// TwinCAT 3 PLC project Test
// ProgramVersion: 3.1.4022.4
// libraries:
//   Tc2_Standard, * (Beckhoff Automation GmbH)
//   Tc2_System, * (Beckhoff Automation GmbH)
//   Tc3_Module, * (Beckhoff Automation GmbH)
//   Marquee,0.5,HiJack Automation
// project tree:
//   FBs/ FB_SignalHandling.TcPOU
//   GVLs/ GVL_General.TcGVL, GVL_Machine.TcGVL, GVL_SignalHanlding.TcGVL, HardwareInput.TcDUT, HardWareIO.TcDUT, HardwareOutput.TcDUT, MachineMode.TcDUT
//   / PlcTask.TcTTO
//   POUs/ LampControl.TcPOU, LinkHWIO.TcPOU, LinkUI.TcPOU, MAIN.TcPOU, ModeManger.TcPOU, SignalHandler.TcPOU
// real-time tasks:
//   TASK PlcTask: cycle T#10ms, priority 20, ADS port 350
// I/O:
//   DEVICE Device 2 (EtherCAT), AmsNetId 192.168.1.105.3.1
//     Term 1 (EK1814) [EK1814 EtherCAT IO-Coupler  (1A E-Bus, 4 Ch. Dig. In, 3ms, 4 Ch. Dig. Out 24V, 0,5A)]
// variable links:
//   Test/Test Instance <-> Device 2 (EtherCAT)/Term 1 (EK1814)
//     PlcTask Inputs/GVL_Machine.HWIO.HWInput.PauseBtn <-> Channel 3/Input
//     PlcTask Inputs/GVL_Machine.HWIO.HWInput.StartBtn <-> Channel 1/Input
//     PlcTask Inputs/GVL_Machine.HWIO.HWInput.StopBtn <-> Channel 2/Input
//     PlcTask Outputs/GVL_Machine.HWIO.HWOutput.Lamp01 <-> Channel 5/Output
//     PlcTask Outputs/GVL_Machine.HWIO.HWOutput.Lamp02 <-> Channel 6/Output
//     PlcTask Outputs/GVL_Machine.HWIO.HWOutput.Lamp03 <-> Channel 7/Output
//     PlcTask Outputs/GVL_Machine.HWIO.HWOutput.Lamp04 <-> Channel 8/Output

CONFIGURATION Test
    RESOURCE PLC ON TwinCAT3
        TASK PlcTask(INTERVAL := T#10ms, PRIORITY := 20);
        PROGRAM MAIN WITH PlcTask : MAIN;
    END_RESOURCE
END_CONFIGURATION

// ---- GVLs/HardwareInput.TcDUT
TYPE HardwareInput :
STRUCT
	StartBtn			AT%I*	 	:BOOL;
	StopBtn				AT%I*	 	:BOOL;
	PauseBtn			AT%I*	 	:BOOL;
END_STRUCT
END_TYPE

// ---- GVLs/HardWareIO.TcDUT
TYPE HardWareIO :
STRUCT
	HWInput			:HardwareInput;
	HWOutput		:HardwareOutput;
END_STRUCT
END_TYPE

// ---- GVLs/HardwareOutput.TcDUT
TYPE HardwareOutput :
STRUCT
	//===============================hardware output===============
	Lamp01			AT %Q* :BOOL;
	Lamp02			AT %Q* :BOOL;
	Lamp03			AT %Q* :BOOL;
	Lamp04			AT %Q* :BOOL;
	//===============================hardware output===============
END_STRUCT
END_TYPE

// ---- GVLs/MachineMode.TcDUT
{attribute 'qualified_only'}
{attribute 'strict'}
TYPE MachineMode :
(
	Idle := 0,
	Auto	:=1,
	Manual	:=2,
	Undefined	:=10
);
END_TYPE

// ---- GVLs/GVL_General.TcGVL
{attribute 'qualified_only'}
VAR_GLOBAL
	
	tDelay					:TIME:= T#1S;
	
	//=====================UI Button=============================
	bStartBtnUI			:BOOL;
	bStopBtnUI			:BOOL;
	bPauseBtnUI			:BOOL;
	//=====================UI Button=============================
	
	btemp		:BOOL;
	//=============Function Blcok instance===================
	fbMarqueeExPause		:FB_MarqueeExPause:=(pLamp01:=ADR(GVL_Machine.HWIO.HWOutput.Lamp01),pLamp02:=ADR(GVL_Machine.HWIO.HWOutput.Lamp02),
												pLamp03:=ADR(GVL_Machine.HWIO.HWOutput.Lamp03),pLamp04:=ADR(GVL_Machine.HWIO.HWOutput.Lamp04),
												pTime:=ADR(GVL_General.tDelay),pPause:=ADR(GVL_SignalHanlding.inPauseBtnHandling.bSignalOutput),
												pStop:=ADR(GVL_Machine.HWIO.HWInput.StopBtn));
	
	
	
END_VAR

// ---- GVLs/GVL_Machine.TcGVL
{attribute 'qualified_only'}
VAR_GLOBAL
	HWIO		:HardWareIO;
	machineMode			:MachineMode;
END_VAR

// ---- GVLs/GVL_SignalHanlding.TcGVL
{attribute 'qualified_only'}
VAR_GLOBAL
	
	//fbPauseUI		:FB_SignalHandling :=(bSignalInput:= GVL_General.bPauseBtnUI);   cannot assigned the signal here.
	fbPauseUI		:FB_SignalHandling;
	
	fbHandleStartBtn		:FB_SignalHandling;
	inPauseBtnHandling	:FB_SignalHandling;
END_VAR

// ---- POUs/MAIN.TcPOU
PROGRAM MAIN
VAR
	
END_VAR


	SignalHandler();
	
//======================Handl the signal from UI=================== 
	LinkUI();
//======================Handl the signal from UI=================== 



//======================Handl the signal from Hardware===================
	LinkHWIO();
//======================Handl the signal from Hardware===================




//====================handle the lights rolling======================
	LampControl();
//====================handle the lights rolling======================

//=========Machine mode selecion================
	ModeManger();
//=========Machine mode selecion================

END_PROGRAM

// ---- POUs/SignalHandler.TcPOU
PROGRAM SignalHandler
VAR
END_VAR

END_PROGRAM

// ---- POUs/LinkUI.TcPOU
PROGRAM LinkUI
VAR
	
END_VAR


//==================Pause button from UI================================
GVL_SignalHanlding.fbPauseUI.bSignalInput := GVL_General.bPauseBtnUI;
GVL_SignalHanlding.fbPauseUI.SignalEnable(bSignalLocalEnable:= TRUE);
GVL_SignalHanlding.fbPauseUI.SetOutput();
//==================Pause button from UI================================

END_PROGRAM

// ---- POUs/LinkHWIO.TcPOU
PROGRAM LinkHWIO
VAR
	
END_VAR

GVL_SignalHanlding.fbHandleStartBtn.bSignalInput := GVL_Machine.HWIO.HWInput.StartBtn OR GVL_SignalHanlding.fbHandleStartBtn.bSignalInput;
GVL_SignalHanlding.fbHandleStartBtn.SignalEnable(bSignalLocalEnable := (GVL_Machine.machineMode = MachineMode.Auto));
GVL_SignalHanlding.fbHandleStartBtn.SetOutput();


//==========Hardware signal inPauseBtn handle==========
GVL_SignalHanlding.inPauseBtnHandling.bSignalInput := ((GVL_Machine.HWIO.HWInput.PauseBtn OR GVL_SignalHanlding.fbPauseUI.bSignalOutput
														 OR GVL_SignalHanlding.inPauseBtnHandling.bSignalInput) AND NOT (GVL_Machine.HWIO.HWInput.StartBtn));
GVL_SignalHanlding.inPauseBtnHandling.SignalEnable(bSignalLocalEnable := (GVL_Machine.machineMode = MachineMode.Auto));
GVL_SignalHanlding.inPauseBtnHandling.SetOutput();
//==========Hardware signal inPause handle==========

END_PROGRAM

// ---- POUs/LampControl.TcPOU
PROGRAM LampControl
VAR
END_VAR

GVL_General.fbMarqueeExPause();

//==========call the "Blinking" method ================================
//GVL_General.fbMarqueeExPause.Blinking(bStart:=GVL_Machine.HWIO.HWInput.StartBtn OR GVL_General.bStartBtnUI );

GVL_General.fbMarqueeExPause.Blinking(bStart:=GVL_SignalHanlding.fbHandleStartBtn.bSignalOutput OR GVL_General.bStartBtnUI );

END_PROGRAM

// ---- POUs/ModeManger.TcPOU
PROGRAM ModeManger
VAR
END_VAR

GVL_Machine.machineMode := MachineMode.Auto;

END_PROGRAM

// ---- FBs/FB_SignalHandling.TcPOU
FUNCTION_BLOCK FB_SignalHandling
VAR_INPUT
	bSignalInput			:BOOL;
END_VAR
VAR_OUTPUT
	bSignalOutput			:BOOL;
END_VAR
VAR
	bLocalEnable		:BOOL;
END_VAR

METHOD SetOutput : BOOL
VAR_INPUT
END_VAR
bSignalOutput := (bLocalEnable AND bSignalInput);
END_METHOD

METHOD SignalEnable : BOOL
VAR_INPUT
	bSignalLocalEnable		:BOOL;
END_VAR
bLocalEnable := bSignalLocalEnable;
END_METHOD

END_FUNCTION_BLOCK
